% RSLogix 500 project I2P Hands-On 4 - Alexander_Loynd.RSS, saved by version 10.00.00.00 %
PROJECT "UNTITLED"    % processor: Bul.1763 MicroLogix 1100 Series B %

PROGRAM FILES
  LAD 2   16 rungs

DATA FILES
  O0 OUTPUT  4 elements
  I1 INPUT  6 elements
  S2 STATUS  66 elements
  B3 BINARY  1 elements
  T4 TIMER  1 elements
  C5 COUNTER  1 elements
  R6 CONTROL  1 elements
  N7 INTEGER  1 elements
  F8 FLOAT  1 elements

LADDER 2
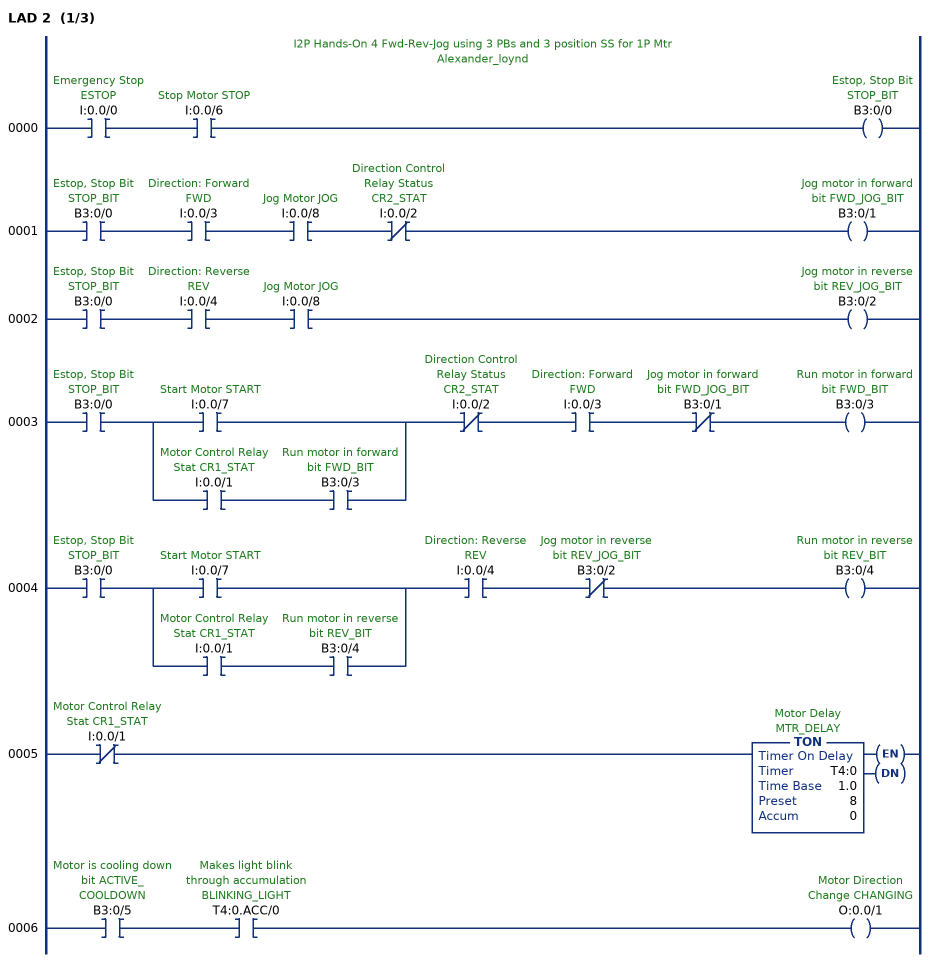
% Rung: 0 %
% I2P Hands-On 4 Fwd-Rev-Jog using 3 PBs and 3 position SS for 1P Mtr
% Alexander_loynd %
SOR XIC I:0.0/0 XIC I:0.0/6 OTE B3:0/0 EOR
%   I:0.0/0  ESTOP  "Emergency Stop" %
%   I:0.0/6  STOP  "Stop Motor" %
%   B3:0/0  STOP_BIT  "Estop, Stop Bit" %
% Rung: 1 %
SOR XIC B3:0/0 XIC I:0.0/3 XIC I:0.0/8 XIO I:0.0/2 OTE B3:0/1 EOR
%   B3:0/0  STOP_BIT  "Estop, Stop Bit" %
%   I:0.0/3  FWD  "Direction: Forward" %
%   I:0.0/8  JOG  "Jog Motor" %
%   I:0.0/2  CR2_STAT  "Direction Control Relay Status" %
%   B3:0/1  FWD_JOG_BIT  "Jog motor in forward bit" %
% Rung: 2 %
SOR XIC B3:0/0 XIC I:0.0/4 XIC I:0.0/8 OTE B3:0/2 EOR
%   B3:0/0  STOP_BIT  "Estop, Stop Bit" %
%   I:0.0/4  REV  "Direction: Reverse" %
%   I:0.0/8  JOG  "Jog Motor" %
%   B3:0/2  REV_JOG_BIT  "Jog motor in reverse bit" %
% Rung: 3 %
SOR XIC B3:0/0 BST XIC I:0.0/7 NXB XIC I:0.0/1 XIC B3:0/3 BND XIO I:0.0/2 XIC I:0.0/3 XIO B3:0/1 OTE B3:0/3 EOR
%   B3:0/0  STOP_BIT  "Estop, Stop Bit" %
%   I:0.0/7  START  "Start Motor" %
%   I:0.0/1  CR1_STAT  "Motor Control Relay Stat" %
%   B3:0/3  FWD_BIT  "Run motor in forward bit" %
%   I:0.0/2  CR2_STAT  "Direction Control Relay Status" %
%   I:0.0/3  FWD  "Direction: Forward" %
%   B3:0/1  FWD_JOG_BIT  "Jog motor in forward bit" %
% Rung: 4 %
SOR XIC B3:0/0 BST XIC I:0.0/7 NXB XIC I:0.0/1 XIC B3:0/4 BND XIC I:0.0/4 XIO B3:0/2 OTE B3:0/4 EOR
%   B3:0/0  STOP_BIT  "Estop, Stop Bit" %
%   I:0.0/7  START  "Start Motor" %
%   I:0.0/1  CR1_STAT  "Motor Control Relay Stat" %
%   B3:0/4  REV_BIT  "Run motor in reverse bit" %
%   I:0.0/4  REV  "Direction: Reverse" %
%   B3:0/2  REV_JOG_BIT  "Jog motor in reverse bit" %
% Rung: 5 %
SOR XIO I:0.0/1 TON T4:0 1.0 8 0 EOR
%   I:0.0/1  CR1_STAT  "Motor Control Relay Stat" %
%   T4:0  MTR_DELAY  "Motor Delay" %
% Rung: 6 %
SOR XIC B3:0/5 XIC T4:0.ACC/0 OTE O:0.0/1 EOR
%   B3:0/5  ACTIVE_COOLDOWN  "Motor is cooling down bit" %
%   T4:0.ACC/0  BLINKING_LIGHT  "Makes light blink through accumulation" %
%   O:0.0/1  CHANGING  "Motor Direction Change" %

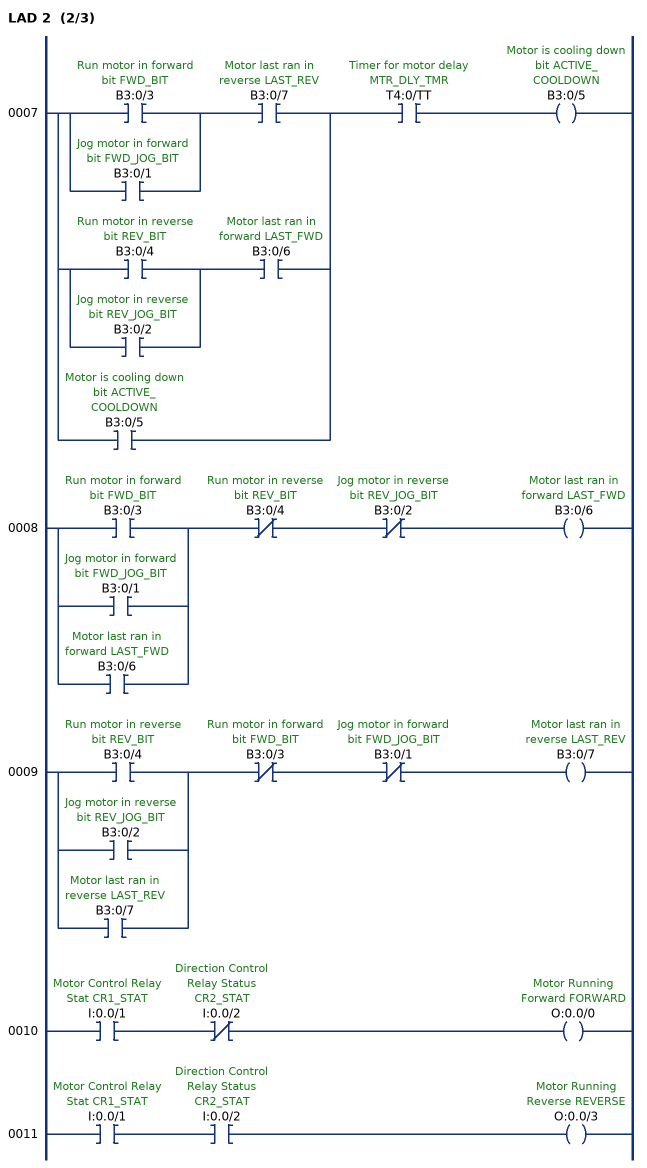
% Rung: 7 %
SOR BST BST BST XIC B3:0/3 NXB XIC B3:0/1 BND XIC B3:0/7 NXB BST XIC B3:0/4 NXB XIC B3:0/2 BND XIC B3:0/6 BND NXB XIC B3:0/5 BND XIC T4:0/TT OTE B3:0/5 EOR
%   B3:0/3  FWD_BIT  "Run motor in forward bit" %
%   B3:0/1  FWD_JOG_BIT  "Jog motor in forward bit" %
%   B3:0/7  LAST_REV  "Motor last ran in reverse" %
%   B3:0/4  REV_BIT  "Run motor in reverse bit" %
%   B3:0/2  REV_JOG_BIT  "Jog motor in reverse bit" %
%   B3:0/6  LAST_FWD  "Motor last ran in forward" %
%   B3:0/5  ACTIVE_COOLDOWN  "Motor is cooling down bit" %
%   T4:0/TT  MTR_DLY_TMR  "Timer for motor delay" %
% Rung: 8 %
SOR BST BST XIC B3:0/3 NXB XIC B3:0/1 BND NXB XIC B3:0/6 BND XIO B3:0/4 XIO B3:0/2 OTE B3:0/6 EOR
%   B3:0/3  FWD_BIT  "Run motor in forward bit" %
%   B3:0/1  FWD_JOG_BIT  "Jog motor in forward bit" %
%   B3:0/6  LAST_FWD  "Motor last ran in forward" %
%   B3:0/4  REV_BIT  "Run motor in reverse bit" %
%   B3:0/2  REV_JOG_BIT  "Jog motor in reverse bit" %
% Rung: 9 %
SOR BST BST XIC B3:0/4 NXB XIC B3:0/2 BND NXB XIC B3:0/7 BND XIO B3:0/3 XIO B3:0/1 OTE B3:0/7 EOR
%   B3:0/4  REV_BIT  "Run motor in reverse bit" %
%   B3:0/2  REV_JOG_BIT  "Jog motor in reverse bit" %
%   B3:0/7  LAST_REV  "Motor last ran in reverse" %
%   B3:0/3  FWD_BIT  "Run motor in forward bit" %
%   B3:0/1  FWD_JOG_BIT  "Jog motor in forward bit" %
% Rung: 10 %
SOR XIC I:0.0/1 XIO I:0.0/2 OTE O:0.0/0 EOR
%   I:0.0/1  CR1_STAT  "Motor Control Relay Stat" %
%   I:0.0/2  CR2_STAT  "Direction Control Relay Status" %
%   O:0.0/0  FORWARD  "Motor Running Forward" %
% Rung: 11 %
SOR XIC I:0.0/1 XIC I:0.0/2 OTE O:0.0/3 EOR
%   I:0.0/1  CR1_STAT  "Motor Control Relay Stat" %
%   I:0.0/2  CR2_STAT  "Direction Control Relay Status" %
%   O:0.0/3  REVERSE  "Motor Running Reverse" %

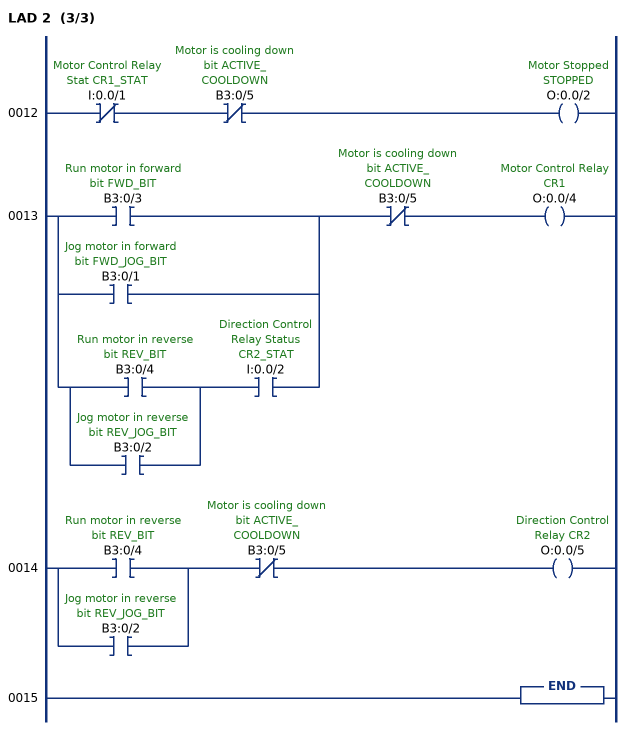
% Rung: 12 %
SOR XIO I:0.0/1 XIO B3:0/5 OTE O:0.0/2 EOR
%   I:0.0/1  CR1_STAT  "Motor Control Relay Stat" %
%   B3:0/5  ACTIVE_COOLDOWN  "Motor is cooling down bit" %
%   O:0.0/2  STOPPED  "Motor Stopped" %
% Rung: 13 %
SOR BST XIC B3:0/3 NXB BST XIC B3:0/1 NXB BST XIC B3:0/4 NXB XIC B3:0/2 BND XIC I:0.0/2 BND BND XIO B3:0/5 OTE O:0.0/4 EOR
%   B3:0/3  FWD_BIT  "Run motor in forward bit" %
%   B3:0/1  FWD_JOG_BIT  "Jog motor in forward bit" %
%   B3:0/4  REV_BIT  "Run motor in reverse bit" %
%   B3:0/2  REV_JOG_BIT  "Jog motor in reverse bit" %
%   I:0.0/2  CR2_STAT  "Direction Control Relay Status" %
%   B3:0/5  ACTIVE_COOLDOWN  "Motor is cooling down bit" %
%   O:0.0/4  CR1  "Motor Control Relay" %
% Rung: 14 %
SOR BST XIC B3:0/4 NXB XIC B3:0/2 BND XIO B3:0/5 OTE O:0.0/5 EOR
%   B3:0/4  REV_BIT  "Run motor in reverse bit" %
%   B3:0/2  REV_JOG_BIT  "Jog motor in reverse bit" %
%   B3:0/5  ACTIVE_COOLDOWN  "Motor is cooling down bit" %
%   O:0.0/5  CR2  "Direction Control Relay" %
% Rung: 15 %
SOR END EOR

DATA TABLE (non-zero values as saved)
DATA T4
% .PRE .ACC %
% T4:0 % 8 0
